(* Schneider Machine Expert - Basic project Questao3.1_FelipeV1_20241008, file version 2.9.0.0 *)
(* ProjectInformations: Name=Novo projeto *)

HARDWARE
  Cpu 0: TM221M16R/G
  EthernetConfiguration: NetworkName=M221, IpAllocationMode=FixedAddress, IpAddress=0.0.0.0, SubnetMask=0.0.0.0
  SerialLineConfiguration: Baud=Baud19200, Parity=ParityEven, DataBits=DataBits8, StopBits=StopBits1, PhysicalMedium=PhysicalMediumRs485, TransmissionMode=TransmissionModeModbusRtu, SlaveId=1, Addressing=SlaveAddressing
  MastTask: UsePeriodScanMode=false, PeriodScan=100
  FastTask: Period=255
  CpuBehavior: StartingMode=StartAsPreviousState, AutoSaveRamOnEeprom=true, WatchdogPeriod=250

SYMBOLS  (address, symbol, comment, settings)
  %I0.0       "A"
  %I0.1       "B"
  %I0.2       "C"
  %I0.3       "D"
  %Q0.1       "Saida P"
  %Q0.2       "Saida M1"
  %Q0.3       "Saida M2"
  %Q0.4       "Saida Alarme"

POU Novo POU
  (* SectionNumber=0 *)

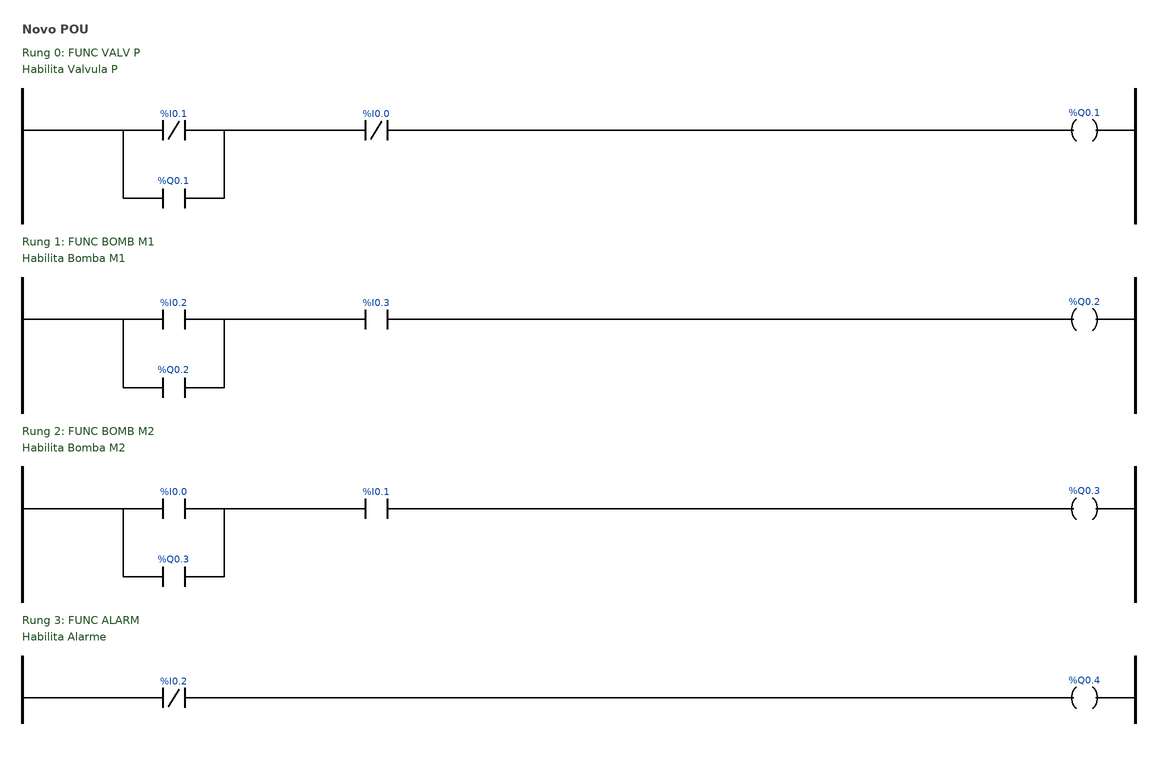

// Rung 0: FUNC VALV P
// Habilita Valvula P
  LD 1
  AND(N %I0.1
  OR %Q0.1
  )
  ANDN %I0.0
  ST %Q0.1
  // as ST:
  //   %Q0.1 := (NOT %I0.1 OR %Q0.1) AND NOT %I0.0;

// Rung 1: FUNC BOMB M1
// Habilita Bomba M1
  LD 1
  AND( %I0.2
  OR %Q0.2
  )
  AND %I0.3
  ST %Q0.2
  // as ST:
  //   %Q0.2 := (%I0.2 OR %Q0.2) AND %I0.3;

// Rung 2: FUNC BOMB M2
// Habilita Bomba M2
  LD 1
  AND( %I0.0
  OR %Q0.3
  )
  AND %I0.1
  ST %Q0.3
  // as ST:
  //   %Q0.3 := (%I0.0 OR %Q0.3) AND %I0.1;

// Rung 3: FUNC ALARM
// Habilita Alarme
  LDN %I0.2
  ST %Q0.4
  // as ST:
  //   %Q0.4 := NOT %I0.2;
